// TIA Portal V19 export
VAR_GLOBAL   // PLC tag table "A0301_COSTANT"
   "%I351.7" AT %I351.7 : Bool;
END_VAR
VAR_GLOBAL CONSTANT   // user constants
   A0301_Distanza_P1toP2 : LReal := 360.0;
   A0301_Distanza_P1toP3 : LReal := 700.0;
   A0301_Distanza_P2toP3 : LReal := 360.0;
   A0301_Distanza_P2toP4 : LReal := 630.0;
   A0301_Distanza_P3toP4 : LReal := 360.0;
   A0301_Tollerance : LReal := 10.0;
END_VAR
